// TIA Portal V19 export
VAR_GLOBAL   // PLC tag table "LB111"
   LB111_Coilcar_Lp_Bwd AT %Q114.7 : Bool;   // 321SH6
   LB111_Coilcar_Lp_Down AT %Q114.5 : Bool;   // 321SH4
   LB111_Coilcar_Lp_Fwd AT %Q114.6 : Bool;   // 321SH5
   LB111_Coilcar_Lp_Up AT %Q114.4 : Bool;   // 321SH3
   LB111_Coilcar_Pb_Bwd AT %I117.1 : Bool;   // 321SH6
   LB111_Coilcar_Pb_Down AT %I116.7 : Bool;   // 321SH4
   LB111_Coilcar_Pb_Fwd AT %I117.0 : Bool;   // 321SH5
   LB111_Coilcar_Pb_Up AT %I116.6 : Bool;   // 321SH3
   LB111_Decoiler_Jaws_Lp_Close AT %Q114.3 : Bool;   // 321SH2
   LB111_Decoiler_Jaws_Lp_Open AT %Q114.2 : Bool;   // 321SH1
   LB111_Decoiler_Jaws_Pb_Close AT %I116.5 : Bool;   // 321SH2
   LB111_Decoiler_Jaws_Pb_Open AT %I116.4 : Bool;   // 321SH1
   LB111_Decoiler_Lp_Bwd AT %Q114.1 : Bool;   // 320SH6
   LB111_Decoiler_Lp_Fwd AT %Q114.0 : Bool;   // 320SH5
   LB111_Decoiler_Pb_Bwd AT %I116.3 : Bool;   // 320SH6
   LB111_Decoiler_Pb_Fwd AT %I116.2 : Bool;   // 320SH5
   LB111_Snubber_Lp_Bwd AT %Q113.7 : Bool;   // 320SH4
   LB111_Snubber_Lp_Down AT %Q113.5 : Bool;   // 320SH2
   LB111_Snubber_Lp_Fwd AT %Q113.6 : Bool;   // 320SH3
   LB111_Snubber_Lp_Up AT %Q113.4 : Bool;   // 320SH1
   LB111_Snubber_Pb_Bwd AT %I116.1 : Bool;   // 320SH4
   LB111_Snubber_Pb_Down AT %I115.7 : Bool;   // 320SH2
   LB111_Snubber_Pb_Fwd AT %I116.0 : Bool;   // 320SH3
   LB111_Snubber_Pb_Up AT %I115.6 : Bool;   // 320SH1
   LB111_Button_L AT %I1027.3 : Bool;   // 103DI3 - 198SB3
   LB111_Button_R AT %I1027.7 : Bool;   // 103DI7 - 198SB4
END_VAR
